PROGRAM UnitTest
VAR
	fbTaskRunner_Test : FB_TaskRunner_Test;
END_VAR

TcUnit.RUN();

END_PROGRAM

(* stored: Version 1.1.0.1, ProductVersion 3.1.4024.15
   POU UnitTest: Id {3459d50f-46c2-4d8b-9955-5e66ae56a75a}, SpecialFunc None *)
